PROGRAM P_init_dauernd
VAR
END_VAR

(* Variablen werden vor jedem Zyklus mit den Werten unten überschrieben *)

(* z.B. Netz_ROT.Parameter.T_Max *)

GA_Global.Zeit_TaskCycle := T#50ms;

END_PROGRAM

(* stored: Version 1.1.0.1, ProductVersion 3.1.4024.9
   POU P_init_dauernd: Id {e1486204-e9dc-46c9-a9f2-3d08451ee3a8}, SpecialFunc None *)
